// FB_Veiligheid.scl
// Veiligheidsverwerking voor automatisch hek
// Verwerkt PBV (persoonsbeveiligingsbumper), VS (veilig sluiten), en sensordefect detectie
// Prioriteit: FAULT > PBV > VS
//
// Versie 0.2: Geconverteerd van FC naar FB voor timer state behoud
//             TON timers voor debounce van alle veiligheidssensoren
//
// NC Sensor logica:
//   i_PBV_BeweegbaarHek: NC, 1 = trigger (bumper geraakt of draadbreuk)
//   i_VS_Voertuig: 0 = geblokkeerd, 1 = intact
//   i_BNS_Open/Dicht: NC, 0 = bereikt, 1 = niet bereikt

FUNCTION_BLOCK "FB_Veiligheid"
{ S7_Optimized_Access := 'TRUE' }
VERSION : 0.2

   VAR_INPUT
      i_PBV_BeweegbaarHek : Bool;   // Persoonsbeveiliging beweegbaar hek (NC: 0=OK, 1=trigger)
      i_VS_Voertuig : Bool;          // Voertuigdetectie lichtsluis (0=onderbroken)
      i_BNS_Open : Bool;             // Benaderingsschakelaar OPEN positie (NC: 0=bereikt)
      i_BNS_Dicht : Bool;            // Benaderingsschakelaar DICHT positie (NC: 0=bereikt)
   END_VAR

   VAR_OUTPUT
      q_PBV_Trigger : Bool;          // PBV geactiveerd (gedebounced, prioriteit toegepast)
      q_VS_Trigger : Bool;           // VS geactiveerd (gedebounced, prioriteit toegepast)
      q_Fault : Bool;                // Sensordefect gedetecteerd (hoogste prioriteit)

      // Combined safety output for state machine
      q_SafetyStop : Bool;           // TRUE = any safety condition active, motor must stop

      // Debug flags (individual active states, before priority masking)
      q_Debug_PBV_Active : Bool;     // Raw debounced PBV state (before priority)
      q_Debug_VS_Active : Bool;      // Raw debounced VS state (before priority)
      q_Debug_Fault_Active : Bool;   // Raw debounced FAULT state
   END_VAR

   VAR
      // Timer instances voor debouncing - state behouden tussen PLC cycles
      m_TON_PBV : TON;               // Timer voor PBV debounce (50ms)
      m_TON_VS : TON;                // Timer voor VS debounce (100ms)
      m_TON_Fault : TON;             // Timer voor FAULT debounce (50ms)

      // Hulpvariabelen voor tussenresultaten
      m_RawFault : Bool;             // Beide eindstanden tegelijk actief
      m_RawVS_Blocked : Bool;        // VS beam onderbroken
   END_VAR

BEGIN
    // =========================================================================
    // STAP 1: DEBOUNCE (uitgevoerd door TON timers)
    // =========================================================================
    // FAULT: beide eindstanden tegelijk actief (NC: 0 = bereikt)
    #m_RawFault := (NOT #i_BNS_Open) AND (NOT #i_BNS_Dicht);
    #m_TON_Fault(IN := #m_RawFault, PT := "DB_Config".Timers.CFG_EndstopDebounceMs);

    // PBV: NC sensor, 1 = trigger (bumper contact of draadbreuk)
    #m_TON_PBV(IN := #i_PBV_BeweegbaarHek, PT := "DB_Config".Timers.CFG_EndstopDebounceMs);

    // VS: 0 = onderbroken (voertuig in lichtsluis)
    #m_RawVS_Blocked := NOT #i_VS_Voertuig;
    #m_TON_VS(IN := #m_RawVS_Blocked, PT := "DB_Config".Safety.CFG_VS_DebounceMs);

    // =========================================================================
    // STAP 2: DEBUG FLAGS (raw debounced, geen prioriteit)
    // =========================================================================
    #q_Debug_Fault_Active := #m_TON_Fault.Q;
    #q_Debug_PBV_Active := #m_TON_PBV.Q;
    #q_Debug_VS_Active := #m_TON_VS.Q;

    // =========================================================================
    // STAP 3: PRIORITEITSLOGICA (SAF-01: FAULT > PBV > VS)
    // =========================================================================
    // Evalueer in prioriteitsvolgorde met masking

    // FAULT: hoogste prioriteit, maskeert alles
    #q_Fault := #m_TON_Fault.Q;

    // PBV: tweede prioriteit, alleen actief als geen FAULT
    #q_PBV_Trigger := #m_TON_PBV.Q AND NOT #q_Fault;

    // VS: laagste prioriteit, alleen actief als geen FAULT en geen PBV
    #q_VS_Trigger := #m_TON_VS.Q AND NOT #q_Fault AND NOT #q_PBV_Trigger;

    // =========================================================================
    // STAP 4: GECOMBINEERDE SAFETY STOP
    // =========================================================================
    // TRUE als ENIGE veiligheidsconditie actief is (na debounce)
    #q_SafetyStop := #q_Fault OR #q_PBV_Trigger OR #q_VS_Trigger;

END_FUNCTION_BLOCK
